(* IEC 61131-3 sources: cds-text-sync-reference-project/project-view/PLC/PLC Logic/ST_Application/03_Object_POU_ST/03_Function, 3 files *)

(* ---- Empty_impementation_fn.st ---- *)
FUNCTION Empty_impementation_fn : BOOL
VAR_INPUT
	SomeBool:BOOL;
END_VAR
VAR
END_VAR

(* ---- fnBEETWEEN.st ---- *)
FUNCTION fnBEETWEEN : BOOL
VAR_INPUT
	iValue : INT;
	iMin : INT;
	iMax : INT;
END_VAR
VAR
END_VAR

// --- implementation ---

fnBEETWEEN := iValue >= iMin AND iValue <= iMax;

(* ---- ST_Function.st ---- *)
FUNCTION ST_Function : BOOL
VAR_INPUT
	rValue : REAL;
	rMin : REAL;
	rMax : REAL;
END_VAR
VAR
END_VAR

// --- implementation ---

IF rValue >= rMin AND rValue <= rMax THEN
	ST_Function := TRUE;
ELSE
	ST_Function := FALSE;//sd
END_IF
